FUNCTION_BLOCK FB_BrakesArm
VAR_IN_OUT
	armSignal : BOOL;
	clkSignal : BOOL;
END_VAR
VAR
	tracker : BOOL;
END_VAR
VAR
END_VAR

//because braking pcb is broken
(*
IF NOT armSignal AND NOT clkSignal AND NOT tracker THEN
	armsignal := TRUE;
	clkSignal := TRUE;
	tracker := TRUE;
ELSIF armSignal AND clkSignal AND tracker THEN
	clkSignal := FALSE;
	tracker := FALSE;
END_IF
*)
GVL_FSM.bbrakes_engageGlobal := TRUE;

END_FUNCTION_BLOCK

(* stored: Version 1.1.0.1
   POU FB_BrakesArm: Id {1a49c53a-438a-46aa-b7dc-e596bb02d16b}, SpecialFunc None *)
